Fanuc KAREL source: kd00018.KL

-- PROVISIONAL review KL for V1013-1; original PC SHA256 e73b40592b3d1396a2a6a4bb789bf262002d9104f57fe6a84c0d381711e70ed6
-- Incomplete behavior may be omitted. Consult companion uncertainty JSON. Do not deploy.
PROGRAM KD00018
%NOLOCKGROUP
VAR
  I : INTEGER
  J : INTEGER
  B : BOOLEAN
  R : REAL
  S : STRING[80]
BEGIN
  -- UNRESOLVED_PC offsets 5-7; opcodes 9D,4D
  -- UNRESOLVED_PC offsets 12-16; opcodes 7F
END KD00018
